FUNCTION_BLOCK EL1889
VAR
	_io : EL1xx9_Data;
	{attribute addProperty Name "WcState"}
	_wcState : WcStateInputToggle;
	{attribute addProperty Name "Info data"}
	_infoData : InfoDataBase;
END_VAR

PROPERTY IO : REFERENCE TO EL1xx9_Data
GET
IO REF= _io;
END_GET
END_PROPERTY

PROPERTY WcState : REFERENCE TO WcStateInputToggle
GET
WcState REF= _wcState;
END_GET
END_PROPERTY

END_FUNCTION_BLOCK

(* stored: Version 1.1.0.1, ProductVersion 3.1.4024.9
   POU EL1889: Id {ecac2d89-7d34-08b3-20f2-590b327d0771}, SpecialFunc None
   Property IO: Id {e99bc72b-c642-0a8c-0dc2-e19279857780}
   Get Get: Id {a721d9f4-c43a-0ae9-281d-ce677d04fbca}
   Property WcState: Id {6f39a7e9-d0fe-0a86-0de6-6ed7e02fcb90}
   Get Get: Id {201543f4-3a70-0b15-0b10-844d0aea9548} *)
